FUNCTION_BLOCK FB_02
VAR_INPUT
END_VAR
VAR_OUTPUT
END_VAR
VAR
END_VAR

END_FUNCTION_BLOCK

(* stored: Version 1.1.0.1, ProductVersion 3.1.4024.12
   POU FB_02: Id {dc912302-708d-4f91-8d4d-dc260435f39e}, SpecialFunc None *)
